// TIA Portal V19 export
FUNCTION_BLOCK "TYPIC_C701_IF_KMO"   // FB102, FBD
TITLE = TYPIC_C701_IF_KMO: Koelmachine
{ S7_Optimized_Access := 'TRUE' }
AUTHOR : OCOTECH
FAMILY : Typical
NAME : C701.715
// Logisch Object Besturing: C701.715
// 
// De interne functie koelmachine verzorgt de interne besturing, bewaking en fysieke aansturing van de koelmachine behorend tot de klimaatinstallatie.
// stored: MemoryReserve 10, SetENOAutomatically false
   VAR_INPUT
      STU_IF_KMO { ExternalAccessible := 'False'; ExternalVisible := 'False'; ExternalWritable := 'False'} : Bool;   // Sturing van de interne functie klimaatregeling (IF), koudevraag voor kring
      IN_TME_IN { ExternalAccessible := 'False'; ExternalVisible := 'False'; ExternalWritable := 'False'} : Real;   // Temperatuurmeting koud water in
      IN_TME_UIT { ExternalAccessible := 'False'; ExternalVisible := 'False'; ExternalWritable := 'False'} : Real;   // Temperatuurmeting koud water uit
      IN_DME { ExternalAccessible := 'False'; ExternalVisible := 'False'; ExternalWritable := 'False'} : Real;   // Drukmeting koelen
      IN_SCF { ExternalAccessible := 'False'; ExternalVisible := 'False'; ExternalWritable := 'False'} : Bool;   // Flowmeting (1 = Flow)
      IN_FB_VGV { ExternalAccessible := 'False'; ExternalVisible := 'False'; ExternalWritable := 'False'} : Bool;   // Feedback sturing vrijgave (1 = Vrijgave)
      IN_AL { ExternalAccessible := 'False'; ExternalVisible := 'False'; ExternalWritable := 'False'} : Bool;   // Algemeen alarm koelmachine (1 = Alarm)
      IN_PMP { ExternalAccessible := 'False'; ExternalVisible := 'False'; ExternalWritable := 'False'} : Bool;   // Status circulatiepomp (1 = Aan)
      IN_AL_PMP { ExternalAccessible := 'False'; ExternalVisible := 'False'; ExternalWritable := 'False'} : Bool;   // Storing circulatiepomp (1 = Storing)
      IN_KLP { ExternalAccessible := 'False'; ExternalVisible := 'False'; ExternalWritable := 'False'} : Bool;   // Status klep (1 = Open)
   END_VAR
   VAR_OUTPUT
      VAR_IF_KMO { ExternalAccessible := 'False'; ExternalVisible := 'False'; ExternalWritable := 'False'} : "C701_VAR_IF_KMO_TYPIC";   // Struct met alle variabelen naar bovenliggende functies
      OUT_VGV { ExternalAccessible := 'False'; ExternalVisible := 'False'; ExternalWritable := 'False'} : Bool;   // Vrijgave koelmachine
      OUT_SWA_TME { ExternalAccessible := 'False'; ExternalVisible := 'False'; ExternalWritable := 'False'} : Real;   // Setpunt temperatuur koelwater
      OUT_KLP { ExternalAccessible := 'False'; ExternalVisible := 'False'; ExternalWritable := 'False'} : Bool;   // Aansturing 2wegklep
   END_VAR
   VAR
      STO { ExternalWritable := 'False'} : Struct   // Storingen
         A001 : Bool;   // Fout temperatuurmeting koelwater in
         A002 : Bool;   // Fout temperatuurmeting koelwater uit
         A003 : Bool;   // Fout drukmeting koelwater
         A004 : Bool;   // Fout flowmeting koelwater
         A005 : Bool;   // Fout algemeen koelmachine
         A006 : Bool;   // Fout circulatiepomp
      END_STRUCT;
      VAR { ExternalWritable := 'False'} : Struct   // Variabelen
         TME_IN : Real;   // Temperatuurmeting koelwater in
         TME_UIT : Real;   // Temperatuurmeting koelwater uit
         DME : Real;   // Drukmeting koelwater
         SWA_TME : Real;   // Setpunt koelwater
      END_STRUCT;
   END_VAR
BEGIN

REGION Network 1: START
END_REGION

REGION Network 2: +++ Metingen +++
   // inlezen van temperaturen en druk.
END_REGION

REGION Network 3: +++ Storingen en meldingen +++
   // aanmaken van storingen en meldingen.
END_REGION

REGION Network 4: Storing A001: Fout temperatuurmeting koelwater in
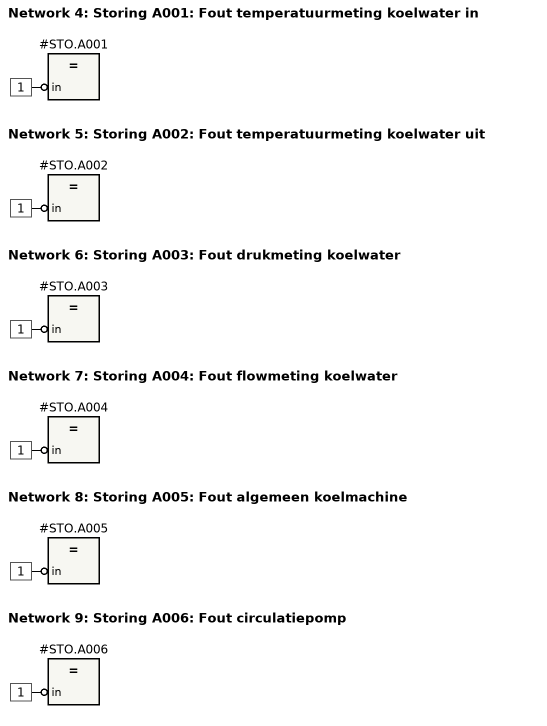
   #STO.A001 := NOT 1;
END_REGION

REGION Network 5: Storing A002: Fout temperatuurmeting koelwater uit
   #STO.A002 := NOT 1;
END_REGION

REGION Network 6: Storing A003: Fout drukmeting koelwater
   #STO.A003 := NOT 1;
END_REGION

REGION Network 7: Storing A004: Fout flowmeting koelwater
   #STO.A004 := NOT 1;
END_REGION

REGION Network 8: Storing A005: Fout algemeen koelmachine
   #STO.A005 := NOT 1;
END_REGION

REGION Network 9: Storing A006: Fout circulatiepomp
   #STO.A006 := NOT 1;
END_REGION

REGION Network 10: +++ Sturingen +++
   // sturing van klep en vrijgave koelmachine in functie van koelvraag.
END_REGION

REGION Network 11 (SCL): EINDE
   // Variabelen van intern scada rakvlak naar outputs copieren
   #VAR_IF_KMO.STO := #STO;
END_REGION
END_FUNCTION_BLOCK
